Staubli VAL3: ServerGet.pgx

public program ServerGet(string& x_sRes (dimensions=1))
  local num l_nIndex
  local num l_nNum[200]
begin
  x_sRes=""

  //从服务器获得字符串
  //  if sioGet(sServer,l_nNum)<0
  //    return
  //  endIf
  wait(sioGet(sServer,l_nNum)>=0)


  //把Acsii转换为字符串
  for l_nIndex=0 to size(l_nNum)-1
    x_sRes=x_sRes+chr(l_nNum[l_nIndex])
  endFor

end
